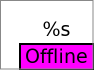
VISUALIZATION Obj_GLP_Status  // 94x70
VAR_INPUT
	sIndex : STRING;
	bAvail : BOOL;
	bOffline : BOOL;
END_VAR
    Rectangle (19,43 75x27), "%s", text list: 'GLP_Available', text index: bAvail
    Rectangle (19,16 75x27), "%s"
    Rectangle (19,43 75x27), "Offline", invisible if: bOffline, text list: 'GLP_Status', text index: bAvail
END_VISUALIZATION

(* stored: Version 1.1.0.1, ProductVersion 3.1.4024.12
   Visu Obj_GLP_Status: Id {4cb1473a-1fd7-435f-969e-a1e35829ffbb} *)
